FUNCTION alg_g_w_w: LREAL
VAR_INPUT
    state: STATE;
END_VAR


        alg_g_w_w := state.curTime;

END_FUNCTION

(* stored: ProductVersion 3.1.0.18, Version 1.1.0.1 *)
